PROGRAM MAIN
VAR
END_VAR

END_PROGRAM

(* stored: Version 1.1.0.1, ProductVersion 3.1.4024.6
   POU MAIN: Id {594bdf20-facb-0c5d-25e5-3d3839948ffc}, SpecialFunc None *)
